PROGRAM P_Demo_F_BA_CountLeapYears
VAR
    argNYear                       : UDINT                          := 0; // nYear
    argNStartYear                  : UDINT                          := 0; // nStartYear
    fnReturn                       : UDINT; // 返回值
END_VAR

// =============================================================================
// Tc3_BA2_Common.F_BA_CountLeapYears 演示程序
// =============================================================================
// 场景：计算从 2000-01-01 到 2025-12-31 之间一共有几个闰年（影响某些累计天数算法）。
//
// 价值：一行 FC 替代 FOR 循环扫描每个年份判断闰年。
//
// 验证：登录 PLC 后，按例程内变量在线写值；监视输出 / 返回值，结合 §1 功能
//       简述的预期行为对照（详见配套 .md 文档 §7 业务场景）。
//
// 验证步骤：
//   1. 右键 PLC 项目下 POUs 文件夹 → Add → Existing Item → 选本 .TcPOU 文件
//   2. 引用 Tc3_BA2_Common（References → Add library）
//   3. 编译 → 登录 → 运行；按上方『验证』指引在线写值观察
// =============================================================================

fnReturn := F_BA_CountLeapYears(
    nYear                    := argNYear,
    nStartYear               := argNStartYear
);

END_PROGRAM

(* stored: Version 1.1.0.1, ProductVersion 3.1.4024.5
   POU P_Demo_F_BA_CountLeapYears: Id {5d5342e9-5a1d-5f7d-9715-93a8f2a6cef2}, SpecialFunc None *)
